(* CODESYS project pwm.2020.08.27.1.v3514.project

Project tree, tasks and I/O mapping:
  MIC7001 : Changsha Xiangji-ARM Cortex A9(xilinx zynq7000)-linux, Changsha Xiangji Hiden Technology Co.Ltd, version 3.5.10.40
    application Application
      libraries: Standard, 3.5.14.0 (System); CAA File, * (CAA Technical Workgroup); CAA Types Extern, * (CAA Technical Workgroup); CAA Callback Extern, * (CAA Technical Workgroup); SysMem, * (System); SysTypes Interfaces, * (System); SysTime, * (System); CAA DTUtil Extern, 3.5.12.0 (CAA Technical Workgroup); cyber gpio, 3.5.10.40 (cyber); CAA Real Time Clock Extern, 3.5.10.0 (CAA Technical Workgroup); CAN API, 1.0.0.3 (3S - Smart Software Solutions GmbH); SysFile, 3.5.15.0 (System); AC_DataLog, 3.5.14.0 (3S - Smart Software Solutions GmbH); CAA SerialCom, 3.5.15.0 (CAA Technical Workgroup); Util, 3.5.15.0 (System); IODrvEtherCAT, 3.5.15.20 (3S - Smart Software Solutions GmbH)
      task Task_10ms (cyclic, interval 10 ms, priority 1) calls prg_pwm_i
      program prg_pwm_i [ST]
      trace Trace (task Task_10ms): prg_pwm_i.pwm_01.real_ma
      PWM/
        function fn_inter_linear [ST]
        function block pwm_ma [ST]
        function block fb_average [ST]
    SoftMotion General Axis Pool
    IoDrvMIC7001 : IoDrvMIC7001, MyCompany, version 19.1.1
        input  Application.prg_pwm_i.pwm_vcc : DWORD  // Ai51_VCC_L
        input  Application.prg_pwm_i.pwm_feedback : DWORD  // Ai53_Pwm-i0
        output Application.prg_pwm_i.pwm_out : DWORD  // PWM_I_0@C33
        unmapped channels: Ai00@C16, Ai01@C28, Ai02@C17, Ai03@C29, Ai04@C30, Ai05@C19, Ai06@C31, Ai07@C20, Ai08@C18, Ai09@D18, Ai10@D20, Ai11@D31, Ai12@D19, Ai13@D30, Ai14@D29, Ai15@D17, Ai16@D28, Ai17@D16, Ai18-Do00@C25, Ai19-Do01@C24, Ai20-Do02@C13, Ai21-Do03@C01, Ai22-Do04@C03, Ai23-Do05@C04, Ai24-Do06@C05, Ai25-Do07@C06, Ai26-Do08@C08, Ai27-Do09@C09, Ai28-Do10@C10, Ai29-Do11@C11, Ai30-Do12@D34, Ai31-Do13@D35, Ai32-Do14@D23, Ai33-Do15@D12, Ai34-Do16@D10, Ai35-Do17@D09, Ai36-Do18@D08, Ai37-Do19@D07, Ai38-Do20@D05, Ai39-Do21@D04,
          Ai40-Do22@D03, Ai41-Do23@D02, Ai42-Do24@C23, Ai43-Do25@C35, Ai44-Do26@D24, Ai45-Do27@D13, Ai46-Ao00@C22, Ai47-Ao01@D14, Ai48_Pi02, Ai49_Out5V, Ai50_VCC, Ai52_VCC_R, Ai54_Pwm-i1, Ai55_Pwm-i2, Ai56_Pwm-i3, Ai57_CPU-T, Ai58_G-x, Ai59_G-y, Ai60_G-z, Ai61-reserved, Ai62-IO-cntr, Ai63-CDS-cntr, Di00-Ai00@C16, Di01-Ai01@C28, Di02-Ai02@C17, Di03-Ai03@C29, Di04-Ai04@C30, Di05-Ai05@C19, Di06-Ai06@C31, Di07-Ai07@C20, Di08-Ai08@C18, Di09-Ai09@D18, Di10-Ai10@D20, Di11-Ai11@D31, Di12-Ai12@D19, Di13-Ai13@D30, Di14-Ai14@D29, Di15-Ai15@D17, Di16-Ai16@D28, Di17-Ai17@D16,
          Di18-Ai18@C25, Di19-Ai19@C24, Di20-Ai20@C13, Di21-Ai21@C01, Di22-Ai22@C03, Di23-Ai23@C04, Di24-Ai24@C05, Di25-Ai25@C06, Di26-Ai26@C08, Di27-Ai27@C09, Di28-Ai28@C10, Di29-Ai29@C11, Di30-Ai30@D34, Di31-Ai31@D35, Di32-Ai32@D23, Di33-Ai33@D12, Di34-Ai34@D10, Di35-Ai35@D09, Di36-Ai36@D08, Di37-Ai37@D07, Di38-Ai38@D05, Di39-Ai39@D04, Di40-Ai40@D03, Di41-Ai41@D02, Di42-Ai42@C23, Di43-Ai43@C35, Di44-Ai44@D24, Di45-Ai45@D13, Di46-Ai46@C22, Di47-Ai47@D14, Di48-Pi00@C15, Di49-Pi01@C14, Di50-Pi02@D22, Di51-Pi03@D21, Di52-reserved, Di53-reserved, Di54-reserved, Di55-reserved, Di56-reserved, Di57-reserved,
          Di58-reserved, Di59-reserved, Di60-reserved, Di61-reserved, Di62-reserved, Di63-reserved, Pi00-Di48@C15, Pi01-Di49@C14, Pi02-Di50@D22, Pi03-Di51@D21, Do00-Ai18@C25, Do01-Ai19@C24, Do02-Ai20@C13, Do03-Ai21@C01, Do04-Ai22@C03, Do05-Ai23@C04, Do06-Ai24@C05, Do07-Ai25@C06, Do08-Ai26@C08, Do09-Ai27@C09, Do10-Ai28@C10, Do11-Ai29@C11, Do12-Ai30@D34, Do13-Ai31@D35, Do14-Ai32@D23, Do15-Ai33@D12, Do16-Ai34@D10, Do17-Ai35@D09, Do18-Ai36@D08, Do19-Ai37@D07, Do20-Ai38@D05, Do21-Ai39@D04, Do22-Ai40@D03, Do23-Ai41@D02, Do24-Ai42@C23, Do25-Ai43@C35, Do26-Ai44@D24, Do27-Ai45@D13, Do28-Pwmi00@C33, Do29-Pwmi01@C34,
          Do30-Pwmi02@D25, Do31-Pwmi03@D26, PWM00@C25, PWM01@C24, PWM02@C13, PWM03@C01, PWM04@C03, PWM05@C04, PWM06@C05, PWM07@C06, PWM08@C08, PWM09@C09, PWM10@C10, PWM11@C11, PWM12@D34, PWM13@D35, PWM14@D23, PWM15@D12, PWM16@D10, PWM17@D09, PWM18@D08, PWM19@D07, PWM20@D05, PWM21@D04, PWM22@D03, PWM23@D02, PWM24@C23, PWM25@C35, PWM26@D24, PWM27@D13, PWM28-Pwmi00@C33, PWM29-Pwmi01@C34, PWM30-Pwmi02@D25, PWM31-Pwmi03@D26, PWM_I_1@C34, PWM_I_2@D25, PWM_I_3@D26, Ao00-Ai46@C22, Ao01-Ai47@D14, LED_run,
          LED_err, LED_usr, ctrl_ai_raw, ctrl_adjust, ctrl_adj0, ctrl_adj1, ctrl_adj2, ctrl_adj3, ctrl_adj4
  text list GlobalTextList
*)

// MIC7001/Application/prg_pwm_i
PROGRAM prg_pwm_i

VAR
	pwm_01:pwm_ma;   //pwm恒流功能块实例，每个电磁阀需要定义一个
	
	pwm_set_ma:DINT := 400;  //输出电流设定值，单位：mA
	pwm_dither_ma : DINT := 0; //颤振电流， 单位：mA

	pwm_feedback:DINT;  //绑定电流反馈端口
	pwm_out:DWORD;      //绑定PWMi输出端口
	pwm_vcc:DWORD;      //绑定VCC_L 或者 VCC_R端口
    
    ton_ma:Standard.TON:=(PT := T#500MS);
END_VAR


ton_ma(IN := NOT ton_ma.Q);
IF ton_ma.Q THEN
    pwm_set_ma := pwm_set_ma + 50; 
    IF pwm_set_ma > 700 THEN
        pwm_set_ma := 300;
	END_IF
END_IF


//当前在5ms的任务中运行，颤振频率为100Hz，如果需要颤振周期为50Hz，可将周期设置为10ms
pwm_01(pwm_set_ma := pwm_set_ma, pwm_feedback := pwm_feedback, vcc := ANY_TO_DINT(pwm_vcc), dither_ma := pwm_dither_ma);

pwm_out := ANY_TO_DWORD(pwm_01.pwm_out);

END_PROGRAM

// MIC7001/Application/PWM/pwm_ma
FUNCTION_BLOCK pwm_ma   //电流型PWM输出功能块，带颤振功能
VAR_INPUT
    enable:BOOL := TRUE;  //使能
	pwm_set_ma:DINT;  //设定输出电流，单位：mA
	pwm_feedback:DINT;   //电流反馈，可直接绑定PWMi对应的AI端口
	dither_ma :DINT := 0;  //设定颤振电流，单位： mA
    
    //以下参数可以根据系统情况修改默认值，运行过程中可以不用设置
	VCC:DINT:=28000;  //电源电压，可直接绑定VCC_L或者VCC_R对应的AI端口,单位：mV
	res_prop_max:DINT:=40;  //比例阀电阻最大值，单位：欧姆
	res_prop_min:DINT:=10;  //比例阀电阻最小值，单位：欧姆
	res_prop_default:DINT := 20;  // 比例阀电阻默认值， 单位：欧姆
END_VAR

VAR_OUTPUT
	pwm_out:DINT;   //PWM输出，可直接绑定PWMi端口
    real_ma:DINT;  // 实际电流
    res_prop_out:REAL := 0; // 根据电流推测出的比例阀电阻值，单位：欧姆
END_VAR

VAR
    old_set_ma : DINT;
	set_ma:DINT;
	
	old_pwm_out:DINT;
	pwm_stable: BOOL;
	
     //电磁阀校准参数，不同的型号可能不同，需要重新校准. 
    arr_in:ARRAY[0..255] OF DINT := [7,   81,  121, 131, 142, 172, 223, 276, 333, 387, 449, 509, 562, 619, 676, 733, 791, 845, 901, 950, 1000, 1100, 1200, 1300, 1400, 1500, 1600, 1700];  // 控制器的反馈电流值 
	arr_out:ARRAY[0..255] OF DINT:= [100, 167, 204, 213, 222, 249, 295, 342, 393, 442, 498, 552, 600, 649, 701, 752, 803, 851, 901, 946,  990, 1078, 1167, 1256, 1345, 1433, 1522, 1609];  // 万用表显示的电流值
	length:DINT := 28;
    
    res_prop:DINT := 0;  // 内部计算用的比例阀电阻值，单位： 毫欧
	dither_phase: BOOL := FALSE;  //颤振相位，为true时加电流， false减电流
    ton_change:Standard.TON := (PT := T#200MS);  // 输出稳定判断定时器， 连续200ms输出变化不大的时候，才进行电磁阀阻值测量
    filter_ma:fb_average;  // 输入电流滤波器
    init:BOOL := FALSE;
END_VAR

IF NOT init THEN
    init := TRUE;
    IF res_prop = 0 THEN
        res_prop := res_prop_default*1000;
	END_IF
END_IF

IF NOT enable OR VCC < 9000 OR pwm_set_ma = 0 THEN
	pwm_out := 0;
	RETURN;
END_IF

// 增加颤振分量
set_ma := pwm_set_ma;
IF dither_ma > 40 THEN  //颤振分量最多40mA
	dither_ma := 40;
END_IF
IF dither_phase THEN
	set_ma := set_ma + dither_ma;
ELSE
	IF set_ma > dither_ma THEN
		set_ma := set_ma - dither_ma;
	ELSE
		set_ma := 0;
	END_IF
END_IF
dither_phase := NOT dither_phase;

pwm_out := set_ma*4096/(VCC*1000/res_prop);
pwm_out := LIMIT(old_pwm_out -100, pwm_out, old_pwm_out+100);
old_pwm_out := pwm_out;

IF  ABS(set_ma - old_set_ma) > 19 THEN
    old_set_ma := set_ma;
    filter_ma.rst := TRUE;
    ton_change(IN := FALSE);
    RETURN;
END_IF

//电磁比例阀反馈电流计算
real_ma := fn_inter_linear(in := pwm_feedback, arr_in := arr_in, arr_out := arr_out, length := length);
filter_ma(X := ANY_TO_REAL(real_ma));
real_ma := ANY_TO_DINT(filter_ma.Y);

ton_change(IN := TRUE);
IF NOT ton_change.Q THEN
    RETURN;
END_IF	

IF    real_ma < set_ma - 100 THEN	res_prop := res_prop + 100;
ELSIF real_ma > set_ma + 100 THEN	res_prop := res_prop - 100;
ELSIF real_ma < set_ma - 60  THEN	res_prop := res_prop + 60;
ELSIF real_ma > set_ma + 60  THEN	res_prop := res_prop - 60;
ELSIF real_ma < set_ma - 30  THEN	res_prop := res_prop + 30;
ELSIF real_ma > set_ma + 30  THEN	res_prop := res_prop - 30;    
ELSIF real_ma < set_ma - 15  THEN	res_prop := res_prop + 10;
ELSIF real_ma > set_ma + 15  THEN	res_prop := res_prop - 10;
ELSIF real_ma < set_ma - 10  THEN	res_prop := res_prop + 3;
ELSIF real_ma > set_ma + 10  THEN	res_prop := res_prop - 3;    
ELSIF real_ma < set_ma - 2   THEN	res_prop := res_prop + 1;
ELSIF real_ma > set_ma + 2   THEN	res_prop := res_prop - 1;
END_IF 

res_prop := LIMIT(res_prop_min*1000, res_prop, res_prop_max*1000);
res_prop_out := ANY_TO_REAL(res_prop)/1000.0;

END_FUNCTION_BLOCK

// MIC7001/Application/PWM/fn_inter_linear
FUNCTION fn_inter_linear : DINT    //线性差值，输入数组需要从小到大排列
VAR_INPUT
	in:DINT;
	arr_in:ARRAY[0..255] OF DINT;
	arr_out:ARRAY[0..255] OF DINT;
	length:DINT;
END_VAR
VAR
	i:DINT;
	out :DINT;
	pos :DINT := 0;
END_VAR

out := 0;
IF length > 256 THEN
	RETURN;
END_IF

IF in <= arr_in[0] THEN
	out := arr_out[0];
	fn_inter_linear := out;
	RETURN;
ELSIF in >= arr_in[length-1] THEN
	out := arr_out[length-1];
	fn_inter_linear := out;
	RETURN;	
END_IF

i := 0;
REPEAT 
	i := i+1;
UNTIL
	in < arr_in[i]
END_REPEAT
pos := i;

fn_inter_linear := (arr_out[i] - arr_out[i-1])*(in - arr_in[i-1])/(arr_in[i]-arr_in[i-1]) + arr_out[i-1];

END_FUNCTION

// MIC7001/Application/PWM/fb_average
FUNCTION_BLOCK fb_average   // 平均值滤波
VAR_INPUT
    x:REAL;
    n:DINT := 10;
    rst:BOOL := FALSE;
END_VAR
VAR_OUTPUT
    y:REAL;
END_VAR
VAR
    buffer:ARRAY[0..32] OF REAL;
    len :DINT ;
    ptr :DINT := 0;
    init :BOOL := FALSE;
    i : DINT;
END_VAR

len := MIN(n, 32);
IF len <2 THEN
    y := x;
    RETURN;
END_IF

IF rst THEN
    init := FALSE;
    rst := FALSE;
END_IF

IF NOT init THEN
    FOR i := 0 TO len-1 DO
        buffer[i] := x;
	END_FOR
    ptr := 0;
    y := x;
    init := TRUE;
    RETURN;
END_IF

y := y + (x - buffer[ptr])/ANY_TO_REAL(len);
buffer[ptr] := x;

ptr := ptr+1;
IF ptr >= len THEN
    ptr := 0;
END_IF

END_FUNCTION_BLOCK
